FUNCTION_BLOCK PayloadCarrier 
VAR_INPUT
END_VAR
VAR_OUTPUT
END_VAR
VAR
	//aPayloads : ARRAY[1..PAYLOAD_TYPE_SIZE-1] OF I_Payload;
	iPayload : I_Payload;
	ePayloadType : E_Payload_Type;
	aGarbageCollection : ARRAY[1..cSizeOfGarbageCollection] OF POINTER TO POINTER TO BYTE;
	nGarbageCollectionCounter : UINT;
	bLock : BOOL;
	bPayloadAssigned : BOOL;
	ePayloadCarrierMode : E_PAYLOAD_CARRIER_MODE;
	pResetKey : POINTER TO BYTE;
END_VAR
VAR CONSTANT
	cSizeOfGarbageCollection : UINT := 10 * ( PAYLOAD_TYPE_SIZE-1 );
END_VAR

METHOD GetPayload : BOOL
VAR_IN_OUT
	pByte : POINTER TO BYTE;
END_VAR

VAR_INPUT
	ePayloadType : E_Payload_Type;
END_VAR
(*
IF 	THIS^.ePayloadType = ePayloadType
	THEN
		GetPayload :=  __QUERYPOINTER(iPayload, pByte);
END_IF
*)


IF 	iPayload <> 0(*aPayloads[ePayloadType] <> 0*)
	AND THIS^.ePayloadType = ePayloadType
	AND nGarbageCollectionCounter <= cSizeOfGarbageCollection
	AND (
			ePayloadCarrierMode = ONE_TO_MANY
			OR 
			(
				ePayloadCarrierMode = ONE_TO_ONE 
				AND NOT bPayloadAssigned
			)
		)
	THEN
	
		bPayloadAssigned := (ePayloadCarrierMode = ONE_TO_ONE); 
		GetPayload :=   __QUERYPOINTER(iPayload , pByte);// __QUERYPOINTER(aPayloads[ePayloadType], pByte);
		IF 	GetPayload
			THEN
			
			nGarbageCollectionCounter := nGarbageCollectionCounter + 1;
			aGarbageCollection[nGarbageCollectionCounter] := ADR(pByte);
			
		END_IF
		
END_IF
END_METHOD

METHOD ResetPayload : BOOL
VAR_INPUT
	pResetKey : POINTER TO BYTE;
END_VAR
VAR
	i: UINT;
END_VAR
IF 	nGarbageCollectionCounter > 0
	AND pResetKey = THIS^.pResetKey
	THEN
	
	FOR i := 1 TO nGarbageCollectionCounter DO
		aGarbageCollection[i]^ := 0;	
		aGarbageCollection[i]:= 0;		
	END_FOR
	
	nGarbageCollectionCounter := 0;
	(*
	FOR i := 1 TO PAYLOAD_TYPE_SIZE-1 DO
		aPayloads[i] := 0;
	END_FOR
	*)
	iPayload := 0;
	bPayloadAssigned := FALSE;
	bLock := FALSE;
	ResetPayload := TRUE;
	
END_IF
END_METHOD

METHOD SetPayload : BOOL
VAR_INPUT
	iPayload : I_Payload; 
	ePayloadType : E_Payload_Type;
	ePayloadCarrierMode : E_PAYLOAD_CARRIER_MODE;
	pResetKey : POINTER TO BYTE;
END_VAR
(*
IF ePayloadType <> NO_PAYLOAD
	THEN
	
	THIS^.iPayload := iPayload;
	THIS^.ePayloadType := ePayloadType;
	
	SetPayload := TRUE;
	
END_IF
*)

IF 	ePayloadType <> NO_PAYLOAD
	AND ePayloadCarrierMode <> NO_PAYLOAD_CARRIER_MODE
	AND bLock = FALSE
	AND pResetKey <> 0
	THEN
	
	this^.pResetKey := pResetKey;
	bLock := TRUE;
	
	THIS^.ePayloadCarrierMode := ePayloadCarrierMode;
	//THIS^.aPayloads[ePayloadType] := iPayload;
	THIS^.iPayload := iPayload;
	THIS^.ePayloadType := ePayloadType;
	SetPayload := TRUE;
	
END_IF
END_METHOD

END_FUNCTION_BLOCK

(* stored: Version 1.1.0.1, ProductVersion 3.1.4024.2
   POU PayloadCarrier: Id {1fa36593-3ecc-43fd-a15b-6576771ee199}, SpecialFunc None
   Method GetPayload: Id {529fe2e9-48db-47b1-b9db-042c523f458f}
   Method ResetPayload: Id {8009174e-f750-493d-a294-b9ad8b678f7e}
   Method SetPayload: Id {1ada05a6-5913-4254-88a8-7e46ea56218a} *)
